// TIA Portal V19 export
TYPE "LAF_typeJobsStatus"
// Status information related to select job
// stored: Access Published
   STRUCT
      activeJobNumber { ExternalWritable := 'False'} : DInt;   // Number of the currently running job
      previousCycleJobNumber { ExternalWritable := 'False'} : DInt;   // Number of the job from the previous CPU cycle
      manualControlEnabled { ExternalWritable := 'False'} : Bool;   // Control via hmiInterface enabled
      memoryJobTime { ExternalAccessible := 'False'; ExternalVisible := 'False'; ExternalWritable := 'False'} : LReal;   // Memory time of the job runtime
   END_STRUCT;
END_TYPE
